SUBAPPLICATION mapping_Uebung_039 (* Spiegelabfolge V2 mit Schrittkette *)
  (* Standard: 61499-2 *)
  (* Version 1.0, 2023-10-23, franz *)
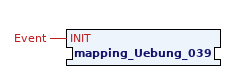
  EVENT_INPUT
    INIT;
  END_EVENT
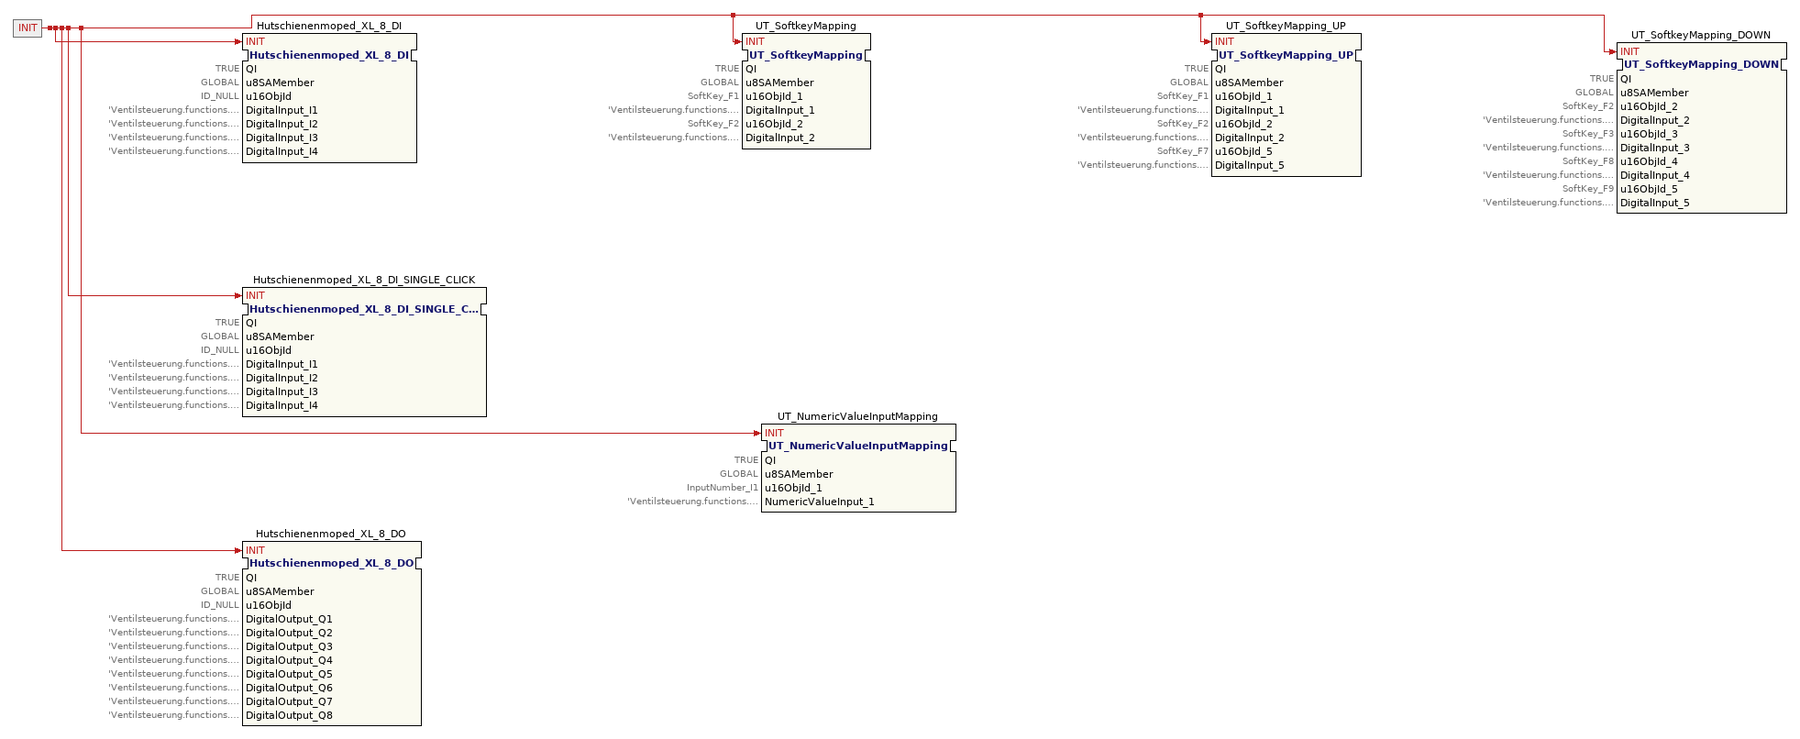
  FBS
    Hutschienenmoped_XL_8_DO : Hutschienenmoped_XL_8_DO(QI := TRUE, u8SAMember := GLOBAL, u16ObjId := ID_NULL, DigitalOutput_Q1 := 'Ventilsteuerung.functions.DigitalOutput_Q1', DigitalOutput_Q2 := 'Ventilsteuerung.functions.DigitalOutput_Q2', DigitalOutput_Q3 := 'Ventilsteuerung.functions.DigitalOutput_Q3', DigitalOutput_Q4 := 'Ventilsteuerung.functions.DigitalOutput_Q4', DigitalOutput_Q5 := 'Ventilsteuerung.functions.DigitalOutput_Q5', DigitalOutput_Q6 := 'Ventilsteuerung.functions.DigitalOutput_Q6', DigitalOutput_Q7 := 'Ventilsteuerung.functions.DigitalOutput_Q7', DigitalOutput_Q8 := 'Ventilsteuerung.functions.DigitalOutput_Q8');
    Hutschienenmoped_XL_8_DI : Hutschienenmoped_XL_8_DI(QI := TRUE, u8SAMember := GLOBAL, u16ObjId := ID_NULL, DigitalInput_I1 := 'Ventilsteuerung.functions.DigitalInput_I1', DigitalInput_I2 := 'Ventilsteuerung.functions.DigitalInput_I2', DigitalInput_I3 := 'Ventilsteuerung.functions.DigitalInput_I3', DigitalInput_I4 := 'Ventilsteuerung.functions.DigitalInput_I4');
    Hutschienenmoped_XL_8_DI_SINGLE_CLICK : Hutschienenmoped_XL_8_DI_SINGLE_CLICK(QI := TRUE, u8SAMember := GLOBAL, u16ObjId := ID_NULL, DigitalInput_I1 := 'Ventilsteuerung.functions.DigitalInput_I1_CLK', DigitalInput_I2 := 'Ventilsteuerung.functions.DigitalInput_I2_CLK', DigitalInput_I3 := 'Ventilsteuerung.functions.DigitalInput_I3_CLK', DigitalInput_I4 := 'Ventilsteuerung.functions.DigitalInput_I4_CLK');
    UT_SoftkeyMapping : UT_SoftkeyMapping(QI := TRUE, u8SAMember := GLOBAL, u16ObjId_1 := SoftKey_F1, DigitalInput_1 := 'Ventilsteuerung.functions.SoftKey_F1', u16ObjId_2 := SoftKey_F2, DigitalInput_2 := 'Ventilsteuerung.functions.SoftKey_F2');
    UT_NumericValueInputMapping : UT_NumericValueInputMapping(QI := TRUE, u8SAMember := GLOBAL, u16ObjId_1 := InputNumber_I1, NumericValueInput_1 := 'Ventilsteuerung.functions.InputNumber_I1');
    UT_SoftkeyMapping_UP : UT_SoftkeyMapping_UP(QI := TRUE, u8SAMember := GLOBAL, u16ObjId_1 := SoftKey_F1, DigitalInput_1 := 'Ventilsteuerung.functions.SoftKey_F1_UP', u16ObjId_2 := SoftKey_F2, DigitalInput_2 := 'Ventilsteuerung.functions.SoftKey_F2_UP', u16ObjId_5 := SoftKey_F7, DigitalInput_5 := 'Ventilsteuerung.functions.SoftKey_F7_UP');
    UT_SoftkeyMapping_DOWN : UT_SoftkeyMapping_DOWN(QI := TRUE, u8SAMember := GLOBAL, u16ObjId_2 := SoftKey_F2, DigitalInput_2 := 'Ventilsteuerung.functions.SoftKey_F2_DOWN', u16ObjId_3 := SoftKey_F3, DigitalInput_3 := 'Ventilsteuerung.functions.SoftKey_F3_DOWN', u16ObjId_4 := SoftKey_F8, DigitalInput_4 := 'Ventilsteuerung.functions.SoftKey_F8_DOWN', u16ObjId_5 := SoftKey_F9, DigitalInput_5 := 'Ventilsteuerung.functions.SoftKey_F9_DOWN');
  END_FBS
  EVENT_CONNECTIONS
    INIT TO Hutschienenmoped_XL_8_DI.INIT;
    INIT TO Hutschienenmoped_XL_8_DO.INIT;
    INIT TO Hutschienenmoped_XL_8_DI_SINGLE_CLICK.INIT;
    INIT TO UT_SoftkeyMapping.INIT;
    INIT TO UT_NumericValueInputMapping.INIT;
    INIT TO UT_SoftkeyMapping_UP.INIT;
    INIT TO UT_SoftkeyMapping_DOWN.INIT;
  END_CONNECTIONS
END_SUBAPPLICATION
